(* IEC 61131-3 sources: LASAL/Class/ST151Base (part 2) *)

//**********************************************************************************************************************************************************
    _InitError:
      eModuleInitState := ERROR;
      if (eInitState <> _InvalidConfguration) then
        eInitState      := _ClientNotready;
      end_if;

//**********************************************************************************************************************************************************

  end_case;

END_FUNCTION

FUNCTION VIRTUAL GLOBAL ST151Base::GetDeviceID
	VAR_OUTPUT
		output 	: UDINT;
	END_VAR

  output := DEVICE_ID_ST151;

END_FUNCTION

FUNCTION VIRTUAL GLOBAL ST151Base::Enable::Write
	VAR_INPUT
		input (EAX) 	: DINT;
	END_VAR
	VAR_OUTPUT
		result (EAX) 	: DINT;
	END_VAR

  if input & AxError then
    input := 0;
  end_if;

  Enable := input;

  sAccesses.sWriteData.ControlWord.SwitchOn := ControlWord.SwitchOn := ControlWord.EnableOperation := to_bool(input);

  if input = 0 then
    SetFreqOut.Write(input:=0);
  end_if;

  result := Enable;

END_FUNCTION

FUNCTION VIRTUAL ST151Base::ReceiveSDOResponse
	VAR_INPUT
		eCommand 	: t_SDIAS_SDO_Cmd;
		hOffset 	: HINT;
		usLength 	: USINT;
		eResult 	: iprStates;
		pResponseBuffer 	: ^USINT;
		ResponseLength 	: USINT;
	END_VAR
	VAR_OUTPUT
		ret_code 	: iprStates;
	END_VAR

  ret_code := SdiasBase::ReceiveSDOResponse(eCommand, hOffset, usLength, eResult, pResponseBuffer, ResponseLength);

  // spi access from baseclass
  if bSDOResponseHandle = TRUE then
    return;
  end_if;

  if eResult = READY then

    case eCommand of
    //**********************************************************************
      SDIAS_SDO_CMD_MEM_WRITE:
        case hOffset of
        //-------------------------------------------------------------
          ST151_ADDR_SDO_1,
          ST151_ADDR_SDO_2,
          ST151_ADDR_SDO_5,
          ST151_ADDR_SDO_6:
            if eResponseState = _wait then
              eResponseState := _valid;
            end_if;
        end_case;

      //**************************************************************************************************************************
      SDIAS_SDO_CMD_MEM_READ:
        case hOffset of
          //***************************************************************************************************
          ST151_ADDR_SDO_1:
            if eResponseState = _wait then
              eResponseState := _valid;
              sReadSDO.SDOData1 := pResponseBuffer^$t_s_ConfigModule1;
            end_if;

          //***************************************************************************************************
          ST151_ADDR_SDO_2:
            if eResponseState = _wait then
              eResponseState := _valid;
              sReadSDO.SDOData2      := pResponseBuffer^$t_s_ConfigModule2;
            end_if;

          //***************************************************************************************************
          ST151_ADDR_SDO_3:
            if eResponseState = _wait then
              eResponseState := _valid;
              sReadSDO.SDOData3      := pResponseBuffer^$t_s_ConfigModule3;
            end_if;

          //***************************************************************************************************
          ST151_ADDR_SDO_4:
            if eResponseState = _wait then
              eResponseState := _valid;
              sReadSDO.SDOData4      := pResponseBuffer^$t_s_ConfigModule4;
            end_if;

          //***************************************************************************************************
          ST151_ADDR_SDO_5:
            if eResponseState = _wait then
              eResponseState := _valid;
              sReadSDO.SDOData5      := pResponseBuffer^$t_s_ConfigModule5;
            end_if;

          //***************************************************************************************************
          ST151_ADDR_SDO_6:
            if eResponseState = _wait then
              eResponseState := _valid;
              sReadSDO.SDOData6      := pResponseBuffer^$t_s_ConfigModule6;
            end_if;
        end_case;

      //**************************************************************************************************************************
      //Control Read
      SDIAS_SDO_CMD_CTRL_READ:
        if hOffset >= ST151_PLL_OFFSET
         & hOffset < (ST151_PLL_OFFSET+sizeof(sPllRegister)) then
          eResponseState := _valid;
          if eResponseState = _wait then
            _memcpy(ptr1:= (#sPllRegister + sSPIReadData.udReadOffset), ptr2:=pResponseBuffer, cntr:=sSPIReadData.udReadLength);
          end_if;
        end_if;

      //**************************************************************************************************************************
      //Control write
      SDIAS_SDO_CMD_CTRL_WRITE:
        if hOffset >= ST151_PLL_OFFSET
         & hOffset < (ST151_PLL_OFFSET+sizeof(sPllRegister)) then
          if eResponseState = _wait then
            eResponseState := _valid;
          end_if;
        end_if;

    end_case;

    if eResponseState <> _valid then
      LogError("@ZZZZ (ST151Base::ReceiveSDOResponse) ERROR in response data of SDO");
      // ERROR was at initialisation
      eInitSSW := _InitError;
    end_if;

  else
    case eCommand of
      SDIAS_SDO_CMD_MEM_WRITE:
        LogError("@ZZZZ (ST151Base::ReceiveSDOResponse) ERROR while writing the sdo data");
      SDIAS_SDO_CMD_MEM_READ:
        LogError("@ZZZZ (ST151Base::ReceiveSDOResponse) ERROR while reading the sdo data");
      SDIAS_SDO_CMD_CTRL_READ:
        LogError("@ZZZZ (ST151Base::ReceiveSDOResponse) Error while reading the pll configuration");
      SDIAS_SDO_CMD_CTRL_WRITE:
        LogError("@ZZZZ (ST151Base::ReceiveSDOResponse) Error while writing the pll configuration");
    end_case;
    // ERROR was at initialisation
    eInitSSW := _InitError;
  end_if;

END_FUNCTION

FUNCTION VIRTUAL GLOBAL ST151Base::Input1LatchedRising::Read
	VAR_OUTPUT
		output (EAX) 	: DINT;
	END_VAR

  //Return Latch
	output := Input1LatchedRising;

  //Reset Latch in next rt-run
  sLatchValues.bsLatchReaded.DigIn1Rise := TRUE;

END_FUNCTION

FUNCTION VIRTUAL GLOBAL ST151Base::Input1LatchedFalling::Read
	VAR_OUTPUT
		output (EAX) 	: DINT;
	END_VAR

  //Return Latch
	output := Input1LatchedFalling;

  //Reset Latch in next rt-run
  sLatchValues.bsLatchReaded.DigIn1Fall := TRUE;

END_FUNCTION

FUNCTION VIRTUAL GLOBAL ST151Base::Input2LatchedRising::Read
	VAR_OUTPUT
		output (EAX) 	: DINT;
	END_VAR

  //Return Latch
	output := Input2LatchedRising;

  //Reset Latch in next rt-run
  sLatchValues.bsLatchReaded.DigIn2Rise := TRUE;

END_FUNCTION

FUNCTION VIRTUAL GLOBAL ST151Base::Input2LatchedFalling::Read
	VAR_OUTPUT
		output (EAX) 	: DINT;
	END_VAR

  //Return Latch
	output := Input2LatchedFalling;

  //Reset Latch in next rt-run
  sLatchValues.bsLatchReaded.DigIn2Fall := TRUE;

END_FUNCTION

FUNCTION VIRTUAL GLOBAL ST151Base::ZPulsLatched::Read
	VAR_OUTPUT
		output (EAX) 	: DINT;
	END_VAR

  //Return Latch
	output := ZPulsLatched;

  //Reset Latch in next rt-run
  sLatchValues.bsLatchReaded.IncZero := TRUE;

END_FUNCTION

FUNCTION VIRTUAL GLOBAL ST151Base::DisconnectEvent
  //Reset DO-Data
  if sAccesses.pWriteData then
    _memset(dest := sAccesses.pWriteData, usByte := 0, cntr := sizeof(sAccesses.pWriteData^));
  end_if;

  //reset online state
  Online  := 0;

  //Call Disconnect of Base-Class
  SdiasBase::DisconnectEvent();

END_FUNCTION

FUNCTION ST151Base::ST151Base
	VAR_OUTPUT
		ret_code 	: ConfStates;
	END_VAR

	ret_code := C_OK;

END_FUNCTION

FUNCTION VIRTUAL ST151Base::GetTaskCfg
	VAR_OUTPUT
		TaskCfg 	: BDINT;
	END_VAR

  TaskCfg := SDIAS_TASK_MASK_RT_PRE OR SDIAS_TASK_MASK_RT_POST OR SDIAS_TASK_MASK_CY;

END_FUNCTION

FUNCTION VIRTUAL GLOBAL ST151Base::ErrorQuit::Write
	VAR_INPUT
		input (EAX) 	: DINT;
	END_VAR
	VAR_OUTPUT
		result (EAX) 	: DINT;
	END_VAR

  result := ErrorQuit := sAccesses.sWriteData.ControlWord.RegenResistorFaultReset := sAccesses.sWriteData.ControlWord.QuitSTOOff := sAccesses.sWriteData.ControlWord.FaultReset := ControlWord.ResetFault := to_bool(input);

END_FUNCTION

FUNCTION VIRTUAL GLOBAL ST151Base::CurrentIncrease::Write
	VAR_INPUT
		input (EAX) 	: DINT;
	END_VAR
	VAR_OUTPUT
		result (EAX) 	: DINT;
	END_VAR

  result := CurrentIncrease := sAccesses.sWriteData.ControlWord.CurrentIncrease := ControlWord.ManufactureSpec1 := to_bool(input);

END_FUNCTION

FUNCTION VIRTUAL GLOBAL ST151Base::ControlWord::Write
	VAR_INPUT
		input (EAX) 	: DS402_Control;
	END_VAR
	VAR_OUTPUT
		result (EAX) 	: DS402_Control;
	END_VAR

  result := ControlWord := input;

  Enable := ControlWord.SwitchOn AND ControlWord.EnableOperation;
  sAccesses.sWriteData.ControlWord.SwitchOn   := to_BOOL(Enable);
  sAccesses.sWriteData.ControlWord.FaultReset := sAccesses.sWriteData.ControlWord.RegenResistorFaultReset := sAccesses.sWriteData.ControlWord.QuitSTOOff := ControlWord.ResetFault;
  CurrentIncrease := sAccesses.sWriteData.ControlWord.CurrentIncrease := ControlWord.ManufactureSpec1;

END_FUNCTION

FUNCTION VIRTUAL GLOBAL ST151Base::SetFreqOut::Write
	VAR_INPUT
		input (EAX) 	: DINT;
	END_VAR
	VAR_OUTPUT
		result (EAX) 	: DINT;
	END_VAR
  VAR
  	dTempInput : DINT;
  END_VAR

  if input <> SetFreqOut then //just do something when the value changed
    dTempInput := input * usCompModeVST;
    if dTempInput > ST151_MAXFREQUENCY_OUT then
      dTempInput := ST151_MAXFREQUENCY_OUT;
    elsif dTempInput < -ST151_MAXFREQUENCY_OUT then
      dTempInput := -ST151_MAXFREQUENCY_OUT;
    end_if;

    //*****************************************************************************
    SetFreqOut := input;

    //Calculate Current
    sAccesses.sWriteData.ControlWord.SwitchMaxCurrent := (abs(input)$UDINT <= udStallCurrentWindow);
    //write act frequency to module
    sAccesses.sWriteData.StepFrequencyReg := dTempInput;

  end_if;

  result := SetFreqOut;

END_FUNCTION

FUNCTION VIRTUAL GLOBAL ST151Base::TargetFreqOut::Write
	VAR_INPUT
		input (EAX) 	: DINT;
	END_VAR
	VAR_OUTPUT
		result (EAX) 	: DINT;
	END_VAR
  VAR
  	dRetCode : DINT;
  END_VAR

  // calculate adaptive microstepping
	TargetFreqOut := input;
  if TargetFreqOut <> -1 then
    //calculate always from zero to target frequency
    dRetCode       := CalcAdaptiveMicroStepping(dTargetFrequency:=TargetFreqOut, dActSetFrequency:=0);
  else
    EnableSteps.Write(input:=EnableSteps+0x800); // +0x800 is just to have a change of the value. It is rejected inside the write()
  end_if;

  if dRetCode = 0 then
    //all ok write setting
  end_if;
	result         := TargetFreqOut;

END_FUNCTION

FUNCTION VIRTUAL GLOBAL ST151Base::HWRampdownDeltaFrequency::Write
	VAR_INPUT
		input (EAX) 	: DINT;
	END_VAR
	VAR_OUTPUT
		result (EAX) 	: DINT;
	END_VAR

  sWriteSDO.SDOData2.HWRampdownDeltaFrequency := input$UINT;
  biReqSDOConfigRdWr.WriteConfigSDO2          := TRUE;
  HWRampdownDeltaFrequency := input;
  result                   := HWRampdownDeltaFrequency;

END_FUNCTION

FUNCTION VIRTUAL GLOBAL ST151Base::HWRampdownDeltaTime::Write
	VAR_INPUT
		input (EAX) 	: DINT;
	END_VAR
	VAR_OUTPUT
		result (EAX) 	: DINT;
	END_VAR

  sWriteSDO.SDOData2.HWRampdownDeltaTime := input$uint;
  biReqSDOConfigRdWr.WriteConfigSDO2     := TRUE;
  HWRampdownDeltaTime := input;
  result              := HWRampdownDeltaTime;

END_FUNCTION

FUNCTION VIRTUAL GLOBAL ST151Base::HWEnableSoftwareRampdown::Write
	VAR_INPUT
		input (EAX) 	: DINT;
	END_VAR
	VAR_OUTPUT
		result (EAX) 	: DINT;
	END_VAR

  HWEnableSoftwareRampdown := input <> 0;
 	result := HWEnableSoftwareRampdown;

END_FUNCTION

FUNCTION ST151Base::SDORdWrData
	VAR_OUTPUT
		dRetCode 	: iprStates;
	END_VAR
  VAR
  	TmpRetcode : iprStates;
  END_VAR

  dRetCode := BUSY;

  case eActSDOConfigRdWr of
    //********************************************************************************************************************************
  	t_e_SDOConfig::_SDOConfig_Idle:
      eActSDOConfigRdWr := SetSDORdWrStep(eActStep:=eActSDOConfigRdWr);

    //********************************************************************************************************************************
  	t_e_SDOConfig::_SDOConfig_Write1:
      case eResponseState of
        _idle:
          biReqSDOConfigRdWr.WriteConfigSDO1  := FALSE;
          bsRespSDOConfigRdWr.WriteConfigSDO1 := FALSE;
          TmpRetcode  := StartWriteSDO(hOffset:=ST151_ADDR_SDO_1, usLength:=sizeof(sWriteSDO.SDOData1), pWriteBuffer:=(#sWriteSDO.SDOData1)$^USINT, eCommand:=SDIAS_SDO_CMD_MEM_WRITE);
          if TmpRetcode = READY then
            udSDOTimeout  := ops.tAbsolute;
            eResponseState:= _wait;
          elsif TmpRetcode = ERROR then
            LogError("@ZZZZ (ST151Base::SDORdWrData) Failed to add write SDO for configuration");
            eActSDOConfigRdWr := _SDOConfig_Error;
          end_if;
          //*****************************************************
        _wait:
          // wait for response
          if ((ops.tAbsolute - udSDOTimeout) > ST151_SDO_RESPONSE_TIMEOUT) then
            LogError("@ZZZZ (ST151Base::SDORdWrData) SDO Response timeout config module");
            eActSDOConfigRdWr := _SDOConfig_Error;
          end_if;
        //*****************************************************
        _valid:
          eActSDOConfigRdWr := SetSDORdWrStep(eActStep:=eActSDOConfigRdWr);
          bsRespSDOConfigRdWr.WriteConfigSDO1 := TRUE;
          eResponseState                      := _idle;
        //*****************************************************
      end_case;

    //********************************************************************************************************************************
  	t_e_SDOConfig::_SDOConfig_Write2:
      case eResponseState of
        _idle:
          biReqSDOConfigRdWr.WriteConfigSDO2  := FALSE;
          bsRespSDOConfigRdWr.WriteConfigSDO2 := FALSE;
          TmpRetcode  := StartWriteSDO(hOffset:=ST151_ADDR_SDO_2, usLength:=sizeof(sWriteSDO.SDOData2), pWriteBuffer:=(#sWriteSDO.SDOData2)$^USINT, eCommand:=SDIAS_SDO_CMD_MEM_WRITE);
          if TmpRetcode = READY then
            udSDOTimeout  := ops.tAbsolute;
            eResponseState:= _wait;
          elsif TmpRetcode = ERROR then
            LogError("@ZZZZ (ST151Base::SDORdWrData) Failed to add write SDO for configuration");
            eActSDOConfigRdWr := _SDOConfig_Error;
          end_if;
          //*****************************************************
        _wait:
          // wait for response
          if ((ops.tAbsolute - udSDOTimeout) > ST151_SDO_RESPONSE_TIMEOUT) then
            LogError("@ZZZZ (ST151Base::SDORdWrData) SDO Response timeout config module");
            eActSDOConfigRdWr := _SDOConfig_Error;
          end_if;
        //*****************************************************
        _valid:
          eActSDOConfigRdWr := SetSDORdWrStep(eActStep:=eActSDOConfigRdWr);
          bsRespSDOConfigRdWr.WriteConfigSDO2 := TRUE;
          eResponseState                      := _idle;
        //*****************************************************
      end_case;

    //********************************************************************************************************************************
  	t_e_SDOConfig::_SDOConfig_Write3:
      //sdo 3 is only read
//      case eResponseState of
//        _idle:
          biReqSDOConfigRdWr.WriteConfigSDO3  := FALSE;
          bsRespSDOConfigRdWr.WriteConfigSDO3 := FALSE;
//          TmpRetcode  := StartWriteSDO(hOffset:=ST151_ADDR_SDO_3, usLength:=sizeof(sWriteSDO.SDOData3), pWriteBuffer:=(#sWriteSDO.SDOData3)$^USINT, eCommand:=SDIAS_SDO_CMD_MEM_WRITE);
//          if TmpRetcode = READY then
//            udSDOTimeout  := ops.tAbsolute;
//            eResponseState:= _wait;
//          elsif TmpRetcode = ERROR then
//            LogError("@ZZZZ (ST151Base::SDORdWrData) Failed to add write SDO for configuration");
//            eActSDOConfigRdWr := _SDOConfig_Error;
//          end_if;
//          //*****************************************************
//        _wait:
//          // wait for response
//          if ((ops.tAbsolute - udSDOTimeout) > ST151_SDO_RESPONSE_TIMEOUT) then
//            LogError("@ZZZZ (ST151Base::SDORdWrData) SDO Response timeout config module");
//            eActSDOConfigRdWr := _SDOConfig_Error;
//          end_if;
//        //*****************************************************
//        _valid:
          eActSDOConfigRdWr := SetSDORdWrStep(eActStep:=eActSDOConfigRdWr);
//          bsRespSDOConfigRdWr.WriteConfigSDO3 := TRUE;
//          eResponseState                      := _idle;
//        //*****************************************************
//      end_case;

    //********************************************************************************************************************************
  	t_e_SDOConfig::_SDOConfig_Write4:
      //sdo 4 is only read
//      case eResponseState of
//        _idle:
          biReqSDOConfigRdWr.WriteConfigSDO4  := FALSE;
          bsRespSDOConfigRdWr.WriteConfigSDO4 := FALSE;
//          TmpRetcode  := StartWriteSDO(hOffset:=ST151_ADDR_SDO_4, usLength:=sizeof(sWriteSDO.SDOData4), pWriteBuffer:=(#sWriteSDO.SDOData4)$^USINT, eCommand:=SDIAS_SDO_CMD_MEM_WRITE);
//          if TmpRetcode = READY then
//            udSDOTimeout  := ops.tAbsolute;
//            eResponseState:= _wait;
//          elsif TmpRetcode = ERROR then
//            LogError("@ZZZZ (ST151Base::SDORdWrData) Failed to add write SDO for configuration");
//            eActSDOConfigRdWr := _SDOConfig_Error;
//          end_if;
//          //*****************************************************
//        _wait:
//          // wait for response
//          if ((ops.tAbsolute - udSDOTimeout) > ST151_SDO_RESPONSE_TIMEOUT) then
//            LogError("@ZZZZ (ST151Base::SDORdWrData) SDO Response timeout config module");
//            eActSDOConfigRdWr := _SDOConfig_Error;
//          end_if;
//        //*****************************************************
//        _valid:
          eActSDOConfigRdWr := SetSDORdWrStep(eActStep:=eActSDOConfigRdWr);
//          bsRespSDOConfigRdWr.WriteConfigSDO4 := TRUE;
//          eResponseState                      := _idle;
//        //*****************************************************
//      end_case;

    //********************************************************************************************************************************
  	t_e_SDOConfig::_SDOConfig_Write5:
      case eResponseState of
        _idle:
          biReqSDOConfigRdWr.WriteConfigSDO5  := FALSE;
          bsRespSDOConfigRdWr.WriteConfigSDO5 := FALSE;
          TmpRetcode  := StartWriteSDO(hOffset:=ST151_ADDR_SDO_5, usLength:=sizeof(sWriteSDO.SDOData5), pWriteBuffer:=(#sWriteSDO.SDOData5)$^USINT, eCommand:=SDIAS_SDO_CMD_MEM_WRITE);
          if TmpRetcode = READY then
            udSDOTimeout  := ops.tAbsolute;
            eResponseState:= _wait;
          elsif TmpRetcode = ERROR then
            LogError("@ZZZZ (ST151Base::SDORdWrData) Failed to add write SDO for configuration");
            eActSDOConfigRdWr := _SDOConfig_Error;
          end_if;
          //*****************************************************
        _wait:
          // wait for response
          if ((ops.tAbsolute - udSDOTimeout) > ST151_SDO_RESPONSE_TIMEOUT) then
            LogError("@ZZZZ (ST151Base::SDORdWrData) SDO Response timeout config module");
            eActSDOConfigRdWr := _SDOConfig_Error;
          end_if;
        //*****************************************************
        _valid:
          eActSDOConfigRdWr := SetSDORdWrStep(eActStep:=eActSDOConfigRdWr);
          bsRespSDOConfigRdWr.WriteConfigSDO5 := TRUE;
          eResponseState                      := _idle;
        //*****************************************************
      end_case;

    //********************************************************************************************************************************
  	t_e_SDOConfig::_SDOConfig_Write6:
      case eResponseState of
        _idle:
          biReqSDOConfigRdWr.WriteConfigSDO6  := FALSE;
          bsRespSDOConfigRdWr.WriteConfigSDO6 := FALSE;
          TmpRetcode  := StartWriteSDO(hOffset:=ST151_ADDR_SDO_6, usLength:=sizeof(sWriteSDO.SDOData6), pWriteBuffer:=(#sWriteSDO.SDOData6)$^USINT, eCommand:=SDIAS_SDO_CMD_MEM_WRITE);
          if TmpRetcode = READY then
            udSDOTimeout  := ops.tAbsolute;
            eResponseState:= _wait;
          elsif TmpRetcode = ERROR then
            LogError("@ZZZZ (ST151Base::SDORdWrData) Failed to add write SDO for configuration");
            eActSDOConfigRdWr := _SDOConfig_Error;
          end_if;
          //*****************************************************
        _wait:
          // wait for response
          if ((ops.tAbsolute - udSDOTimeout) > ST151_SDO_RESPONSE_TIMEOUT) then
            LogError("@ZZZZ (ST151Base::SDORdWrData) SDO Response timeout config module");
            eActSDOConfigRdWr := _SDOConfig_Error;
          end_if;
        //*****************************************************
        _valid:
          eActSDOConfigRdWr := SetSDORdWrStep(eActStep:=eActSDOConfigRdWr);
          bsRespSDOConfigRdWr.WriteConfigSDO6 := TRUE;
          eResponseState                      := _idle;
        //*****************************************************
      end_case;

    //********************************************************************************************************************************
  	t_e_SDOConfig::_SDOConfig_Read1:
      case eResponseState of
        _idle:
          biReqSDOConfigRdWr.ReadConfigSDO1  := FALSE;
          bsRespSDOConfigRdWr.ReadConfigSDO1 := FALSE;
          TmpRetcode  := StartReadSDO(hOffset:=ST151_ADDR_SDO_1, usLength:=sizeof(sReadSDO.SDOData1), eCommand:=SDIAS_SDO_CMD_MEM_READ);
          if TmpRetcode = READY then
            udSDOTimeout  := ops.tAbsolute;
            eResponseState:= _wait;
          elsif TmpRetcode = ERROR then
            LogError("@ZZZZ (ST151Base::SDORdWrData) Failed to add SDO for read of configuration");
            eActSDOConfigRdWr := _SDOConfig_Error;
          end_if;
          //*****************************************************
        _wait:
          // wait for response
          if ((ops.tAbsolute - udSDOTimeout) > ST151_SDO_RESPONSE_TIMEOUT) then
            LogError("@ZZZZ (ST151Base::SDORdWrData) SDO Response timeout config module");
            eActSDOConfigRdWr := _SDOConfig_Error;
          end_if;
        //*****************************************************
        _valid:
          eActSDOConfigRdWr := SetSDORdWrStep(eActStep:=eActSDOConfigRdWr);
          bsRespSDOConfigRdWr.ReadConfigSDO1  := TRUE;
          eResponseState                      := _idle;
        //*****************************************************
      end_case;

    //********************************************************************************************************************************
  	t_e_SDOConfig::_SDOConfig_Read2:
      case eResponseState of
        _idle:
          biReqSDOConfigRdWr.ReadConfigSDO2  := FALSE;
          bsRespSDOConfigRdWr.ReadConfigSDO2 := FALSE;
          TmpRetcode  := StartReadSDO(hOffset:=ST151_ADDR_SDO_2, usLength:=sizeof(sReadSDO.SDOData2), eCommand:=SDIAS_SDO_CMD_MEM_READ);
          if TmpRetcode = READY then
            udSDOTimeout  := ops.tAbsolute;
            eResponseState:= _wait;
          elsif TmpRetcode = ERROR then
            LogError("@ZZZZ (ST151Base::SDORdWrData) Failed to add SDO for read of configuration");
            eActSDOConfigRdWr := _SDOConfig_Error;
          end_if;
          //*****************************************************
        _wait:
          // wait for response
          if ((ops.tAbsolute - udSDOTimeout) > ST151_SDO_RESPONSE_TIMEOUT) then
            LogError("@ZZZZ (ST151Base::SDORdWrData) SDO Response timeout config module");
            eActSDOConfigRdWr := _SDOConfig_Error;
          end_if;
        //*****************************************************
        _valid:
          eActSDOConfigRdWr := SetSDORdWrStep(eActStep:=eActSDOConfigRdWr);
          bsRespSDOConfigRdWr.ReadConfigSDO2  := TRUE;
          eResponseState                      := _idle;
        //*****************************************************
      end_case;

    //********************************************************************************************************************************
  	t_e_SDOConfig::_SDOConfig_Read3:
      case eResponseState of
        _idle:
          biReqSDOConfigRdWr.ReadConfigSDO3  := FALSE;
          bsRespSDOConfigRdWr.ReadConfigSDO3 := FALSE;
          TmpRetcode  := StartReadSDO(hOffset:=ST151_ADDR_SDO_3, usLength:=sizeof(sReadSDO.SDOData3), eCommand:=SDIAS_SDO_CMD_MEM_READ);
          if TmpRetcode = READY then
            //save the actual latched values
            sLatchValues.bsValidISyncValue     := sLatchValues.bsActiveISyncValue;
            sLatchValues.bResetActiveSyncValue := TRUE;
            udSDOTimeout  := ops.tAbsolute;
            eResponseState:= _wait;
          elsif TmpRetcode = ERROR then
            LogError("@ZZZZ (ST151Base::SDORdWrData) Failed to add SDO for read of configuration");
            eActSDOConfigRdWr := _SDOConfig_Error;
          end_if;
          //*****************************************************
        _wait:
          // wait for response
          if ((ops.tAbsolute - udSDOTimeout) > ST151_SDO_RESPONSE_TIMEOUT) then
            LogError("@ZZZZ (ST151Base::SDORdWrData) SDO Response timeout config module");
            eActSDOConfigRdWr := _SDOConfig_Error;
          end_if;
        //*****************************************************
        _valid:
          eActSDOConfigRdWr := SetSDORdWrStep(eActStep:=eActSDOConfigRdWr);
          bsRespSDOConfigRdWr.ReadConfigSDO3  := TRUE;
          eResponseState                      := _idle;
        //*****************************************************
      end_case;

    //********************************************************************************************************************************
  	t_e_SDOConfig::_SDOConfig_Read4:
      case eResponseState of
        _idle:
          biReqSDOConfigRdWr.ReadConfigSDO4  := FALSE;
          bsRespSDOConfigRdWr.ReadConfigSDO4 := FALSE;
          TmpRetcode  := StartReadSDO(hOffset:=ST151_ADDR_SDO_4, usLength:=sizeof(sReadSDO.SDOData4), eCommand:=SDIAS_SDO_CMD_MEM_READ);
          if TmpRetcode = READY then
            //save the actual latched values
            sLatchValues.bsValidISyncValue     := sLatchValues.bsActiveISyncValue;
            sLatchValues.bResetActiveSyncValue := TRUE;
            udSDOTimeout  := ops.tAbsolute;
            eResponseState:= _wait;
          elsif TmpRetcode = ERROR then
            LogError("@ZZZZ (ST151Base::SDORdWrData) Failed to add SDO for read of configuration");
            eActSDOConfigRdWr := _SDOConfig_Error;
          end_if;
          //*****************************************************
        _wait:
          // wait for response
          if ((ops.tAbsolute - udSDOTimeout) > ST151_SDO_RESPONSE_TIMEOUT) then
            LogError("@ZZZZ (ST151Base::SDORdWrData) SDO Response timeout config module");
            eActSDOConfigRdWr := _SDOConfig_Error;
          end_if;
        //*****************************************************
        _valid:
          eActSDOConfigRdWr := SetSDORdWrStep(eActStep:=eActSDOConfigRdWr);
          bsRespSDOConfigRdWr.ReadConfigSDO4  := TRUE;
          eResponseState                      := _idle;
        //*****************************************************
      end_case;

    //********************************************************************************************************************************
  	t_e_SDOConfig::_SDOConfig_Read5:
      case eResponseState of
        _idle:
          biReqSDOConfigRdWr.ReadConfigSDO5  := FALSE;
          bsRespSDOConfigRdWr.ReadConfigSDO5 := FALSE;
          TmpRetcode  := StartReadSDO(hOffset:=ST151_ADDR_SDO_5, usLength:=sizeof(sReadSDO.SDOData5), eCommand:=SDIAS_SDO_CMD_MEM_READ);
          if TmpRetcode = READY then
            udSDOTimeout  := ops.tAbsolute;
            eResponseState:= _wait;
          elsif TmpRetcode = ERROR then
            LogError("@ZZZZ (ST151Base::SDORdWrData) Failed to add SDO for read of configuration");
            eActSDOConfigRdWr := _SDOConfig_Error;
          end_if;
          //*****************************************************
        _wait:
          // wait for response
          if ((ops.tAbsolute - udSDOTimeout) > ST151_SDO_RESPONSE_TIMEOUT) then
            LogError("@ZZZZ (ST151Base::SDORdWrData) SDO Response timeout config module");
            eActSDOConfigRdWr := _SDOConfig_Error;
          end_if;
        //*****************************************************
        _valid:
          eActSDOConfigRdWr := SetSDORdWrStep(eActStep:=eActSDOConfigRdWr);
          bsRespSDOConfigRdWr.ReadConfigSDO5  := TRUE;
          eResponseState                      := _idle;
        //*****************************************************
      end_case;

    //********************************************************************************************************************************
  	t_e_SDOConfig::_SDOConfig_Read6:
      case eResponseState of
        _idle:
          biReqSDOConfigRdWr.ReadConfigSDO6  := FALSE;
          bsRespSDOConfigRdWr.ReadConfigSDO6 := FALSE;
          TmpRetcode  := StartReadSDO(hOffset:=ST151_ADDR_SDO_6, usLength:=sizeof(sReadSDO.SDOData6), eCommand:=SDIAS_SDO_CMD_MEM_READ);
          if TmpRetcode = READY then
            udSDOTimeout  := ops.tAbsolute;
            eResponseState:= _wait;
          elsif TmpRetcode = ERROR then
            LogError("@ZZZZ (ST151Base::SDORdWrData) Failed to add SDO for read of configuration");
            eActSDOConfigRdWr := _SDOConfig_Error;
          end_if;
          //*****************************************************
        _wait:
          // wait for response
          if ((ops.tAbsolute - udSDOTimeout) > ST151_SDO_RESPONSE_TIMEOUT) then
            LogError("@ZZZZ (ST151Base::SDORdWrData) SDO Response timeout config module");
            eActSDOConfigRdWr := _SDOConfig_Error;
          end_if;
        //*****************************************************
        _valid:
          eActSDOConfigRdWr := SetSDORdWrStep(eActStep:=eActSDOConfigRdWr);
          bsRespSDOConfigRdWr.ReadConfigSDO6  := TRUE;
          eResponseState                      := _idle;
        //*****************************************************
      end_case;

    //********************************************************************************************************************************
  	t_e_SDOConfig::_SDOConfig_Finished:
      //all ok sdo config is finished
      dRetCode          := READY;
      usSDORetrys       := 0;
      eActSDOConfigRdWr := _SDOConfig_Idle;

    //********************************************************************************************************************************
  	t_e_SDOConfig::_SDOConfig_Error:
      dRetCode          := ERROR;
      usSDORetrys       += 1;
      if usSDORetrys < ST151_SDO_MAX_RETRYS then
        eActSDOConfigRdWr := _SDOConfig_Idle;
      end_if;
      eResponseState    := _idle;

  end_case;

END_FUNCTION

FUNCTION VIRTUAL GLOBAL ST151Base::FrequLimitIncrease2to1::Write
	VAR_INPUT
		input (EAX) 	: UDINT;
	END_VAR
	VAR_OUTPUT
		result (EAX) 	: UDINT;
	END_VAR
  VAR
    siActArrayEntry : SINT;
  END_VAR

  siActArrayEntry := 0;
  //calculate compatibility mode if client is set
  input *= usCompModeVST;

   // Check for max frequency limit
  if input > ST151_MAXFREQUENCY_OUT then
    input := ST151_MAXFREQUENCY_OUT;
  end_if;

  if aFrequencyLimit[siActArrayEntry].LimitIncrease <> input then //do we have a new value?
    //Save Input
    FrequLimitIncrease2to1 := input / usCompModeVST;

    aFrequencyLimit[siActArrayEntry].LimitIncrease := input;
    FrequLimitDecrease1to2.Write(input:=FrequLimitDecrease1to2);

    if aFrequencyLimit[siActArrayEntry].LimitIncrease <> sWriteSDO.SDOData1.FrequLimitRising2 then //do we have a new value?
      //Set new Limit
      sWriteSDO.SDOData1.FrequLimitRising2 := aFrequencyLimit[siActArrayEntry].LimitIncrease;
      biReqSDOConfigRdWr.WriteConfigSDO1   := TRUE;
    end_if;
  end_if;

  result := FrequLimitIncrease2to1;

END_FUNCTION

FUNCTION VIRTUAL GLOBAL ST151Base::FrequLimitIncrease4to2::Write
	VAR_INPUT
		input (EAX) 	: UDINT;
	END_VAR
	VAR_OUTPUT
		result (EAX) 	: UDINT;
	END_VAR
  VAR
    siActArrayEntry : SINT;
  END_VAR

  siActArrayEntry := 1;
  //calculate compatibility mode if client is set
  input *= usCompModeVST;

   // Check for max frequency limit
  if input > ST151_MAXFREQUENCY_OUT then
    input := ST151_MAXFREQUENCY_OUT;
  end_if;

  if aFrequencyLimit[siActArrayEntry].LimitIncrease <> input then //do we have a new value?
    //Save Input
    FrequLimitIncrease4to2 := input / usCompModeVST;

    aFrequencyLimit[siActArrayEntry].LimitIncrease := input;
    FrequLimitDecrease2to4.Write(input:=FrequLimitDecrease2to4);

    if aFrequencyLimit[siActArrayEntry].LimitIncrease <> sWriteSDO.SDOData1.FrequLimitRising4 then //do we have a new value?
      //Set new Limit
      sWriteSDO.SDOData1.FrequLimitRising4 := aFrequencyLimit[siActArrayEntry].LimitIncrease;
      biReqSDOConfigRdWr.WriteConfigSDO1   := TRUE;
    end_if;
  end_if;

  result := FrequLimitIncrease4to2;

END_FUNCTION

FUNCTION VIRTUAL GLOBAL ST151Base::FrequLimitIncrease8to4::Write
	VAR_INPUT
		input (EAX) 	: UDINT;
	END_VAR
	VAR_OUTPUT
		result (EAX) 	: UDINT;
	END_VAR
  VAR
    siActArrayEntry : SINT;
  END_VAR

  siActArrayEntry := 2;
  //calculate compatibility mode if client is set
  input *= usCompModeVST;

   // Check for max frequency limit
  if input > ST151_MAXFREQUENCY_OUT then
    input := ST151_MAXFREQUENCY_OUT;
  end_if;

  if aFrequencyLimit[siActArrayEntry].LimitIncrease <> input then //do we have a new value?
    //Save Input
    FrequLimitIncrease8to4 := input / usCompModeVST;

    aFrequencyLimit[siActArrayEntry].LimitIncrease := input;
    FrequLimitDecrease4to8.Write(input:=FrequLimitDecrease4to8);

    if aFrequencyLimit[siActArrayEntry].LimitIncrease <> sWriteSDO.SDOData1.FrequLimitRising8 then //do we have a new value?
      //Set new Limit
      sWriteSDO.SDOData1.FrequLimitRising8 := aFrequencyLimit[siActArrayEntry].LimitIncrease;
      biReqSDOConfigRdWr.WriteConfigSDO1   := TRUE;
    end_if;
  end_if;

  result := FrequLimitIncrease8to4;

END_FUNCTION

FUNCTION VIRTUAL GLOBAL ST151Base::FrequLimitIncrease16to8::Write
	VAR_INPUT
		input (EAX) 	: UDINT;
	END_VAR
	VAR_OUTPUT
		result (EAX) 	: UDINT;
	END_VAR
  VAR
    siActArrayEntry : SINT;
  END_VAR

  siActArrayEntry := 3;
  //calculate compatibility mode if client is set
  input *= usCompModeVST;

   // Check for max frequency limit
  if input > ST151_MAXFREQUENCY_OUT then
    input := ST151_MAXFREQUENCY_OUT;
  end_if;

  if aFrequencyLimit[siActArrayEntry].LimitIncrease <> input then //do we have a new value?
    //Save Input
    FrequLimitIncrease16to8 := input / usCompModeVST;

    aFrequencyLimit[siActArrayEntry].LimitIncrease := input;
    FrequLimitDecrease8to16.Write(input:=FrequLimitDecrease8to16);

    if aFrequencyLimit[siActArrayEntry].LimitIncrease <> sWriteSDO.SDOData1.FrequLimitRising16 then //do we have a new value?
      //Set new Limit
      sWriteSDO.SDOData1.FrequLimitRising16 := aFrequencyLimit[siActArrayEntry].LimitIncrease;
      biReqSDOConfigRdWr.WriteConfigSDO1    := TRUE;
    end_if;
  end_if;

  result := FrequLimitIncrease16to8;

END_FUNCTION

FUNCTION VIRTUAL GLOBAL ST151Base::FrequLimitIncrease32to16::Write
	VAR_INPUT
		input (EAX) 	: UDINT;
	END_VAR
	VAR_OUTPUT
		result (EAX) 	: UDINT;
	END_VAR
  VAR
    siActArrayEntry : SINT;
  END_VAR

  siActArrayEntry := 4;
  //calculate compatibility mode if client is set
  input *= usCompModeVST;

   // Check for max frequency limit
  if input > ST151_MAXFREQUENCY_OUT then
    input := ST151_MAXFREQUENCY_OUT;
  end_if;

  if aFrequencyLimit[siActArrayEntry].LimitIncrease <> input then //do we have a new value?
    //Save Input
    FrequLimitIncrease32to16 := input / usCompModeVST;

    aFrequencyLimit[siActArrayEntry].LimitIncrease := input;
    FrequLimitDecrease16to32.Write(input:=FrequLimitDecrease16to32);

    if aFrequencyLimit[siActArrayEntry].LimitIncrease <> sWriteSDO.SDOData1.FrequLimitRising32 then //do we have a new value?
      //Set new Limit
      sWriteSDO.SDOData1.FrequLimitRising32 := aFrequencyLimit[siActArrayEntry].LimitIncrease;
      biReqSDOConfigRdWr.WriteConfigSDO1    := TRUE;
    end_if;
  end_if;

  result := FrequLimitIncrease32to16;

END_FUNCTION

FUNCTION VIRTUAL GLOBAL ST151Base::FrequLimitIncrease64to32::Write
	VAR_INPUT
		input (EAX) 	: UDINT;
	END_VAR
	VAR_OUTPUT
		result (EAX) 	: UDINT;
	END_VAR
  VAR
    siActArrayEntry : SINT;
  END_VAR

  siActArrayEntry := 5;
  //calculate compatibility mode if client is set
  input *= usCompModeVST;

   // Check for max frequency limit
  if input > ST151_MAXFREQUENCY_OUT then
    input := ST151_MAXFREQUENCY_OUT;
  end_if;

  if aFrequencyLimit[siActArrayEntry].LimitIncrease <> input then //do we have a new value?
    //Save Input
    FrequLimitIncrease64to32 := input / usCompModeVST;

    aFrequencyLimit[siActArrayEntry].LimitIncrease := input;
    FrequLimitDecrease32to64.Write(input:=FrequLimitDecrease32to64);

    if aFrequencyLimit[siActArrayEntry].LimitIncrease <> sWriteSDO.SDOData1.FrequLimitRising64 then //do we have a new value?
      //Set new Limit
      sWriteSDO.SDOData1.FrequLimitRising64 := aFrequencyLimit[siActArrayEntry].LimitIncrease;
      biReqSDOConfigRdWr.WriteConfigSDO1    := TRUE;
    end_if;
  end_if;

  result := FrequLimitIncrease64to32;

END_FUNCTION

FUNCTION VIRTUAL GLOBAL ST151Base::FrequLimitDecrease1to2::Write
	VAR_INPUT
		input (EAX) 	: UDINT;
	END_VAR
	VAR_OUTPUT
		result (EAX) 	: UDINT;
	END_VAR
  VAR
    siActArrayEntry : SINT;
  END_VAR

  siActArrayEntry := 0;
  //calculate compatibility mode if client is set
  input *= usCompModeVST;

   // Check for max frequency limit
  if input > ST151_MAXFREQUENCY_OUT then
    input := ST151_MAXFREQUENCY_OUT;
  end_if;
  //Save Input
  FrequLimitDecrease1to2 := input / usCompModeVST;

  if input <> ST151_AUTOSET_FREQUENCYLIMIT then
    aFrequencyLimit[siActArrayEntry].LimitDecrease := input;
  else
    CalcSimpleMode();
  end_if;

  if aFrequencyLimit[siActArrayEntry].LimitDecrease <> sWriteSDO.SDOData5.FrequLimitFalling1to2 then //do we have a new value?
    //Set new Limit
    sWriteSDO.SDOData5.FrequLimitFalling1to2 := aFrequencyLimit[siActArrayEntry].LimitDecrease;
    biReqSDOConfigRdWr.WriteConfigSDO5       := TRUE;
  end_if;

  result := FrequLimitDecrease1to2;

END_FUNCTION

FUNCTION VIRTUAL GLOBAL ST151Base::FrequLimitDecrease2to4::Write
	VAR_INPUT
		input (EAX) 	: UDINT;
	END_VAR
	VAR_OUTPUT
		result (EAX) 	: UDINT;
	END_VAR
  VAR
    siActArrayEntry : SINT;
  END_VAR

  siActArrayEntry := 1;
  //calculate compatibility mode if client is set
  input *= usCompModeVST;

   // Check for max frequency limit
  if input > ST151_MAXFREQUENCY_OUT then
    input := ST151_MAXFREQUENCY_OUT;
  end_if;
  //Save Input
  FrequLimitDecrease2to4 := input / usCompModeVST;

  if input <> ST151_AUTOSET_FREQUENCYLIMIT then
    aFrequencyLimit[siActArrayEntry].LimitDecrease := input;
  else
    CalcSimpleMode();
  end_if;
  if aFrequencyLimit[siActArrayEntry].LimitDecrease <> sWriteSDO.SDOData5.FrequLimitFalling2to4 then //do we have a new value?
    //Set new Limit
    sWriteSDO.SDOData5.FrequLimitFalling2to4 := aFrequencyLimit[siActArrayEntry].LimitDecrease;
    biReqSDOConfigRdWr.WriteConfigSDO5       := TRUE;
  end_if;

  result := FrequLimitDecrease2to4;

END_FUNCTION

FUNCTION VIRTUAL GLOBAL ST151Base::FrequLimitDecrease4to8::Write
	VAR_INPUT
		input (EAX) 	: UDINT;
	END_VAR
	VAR_OUTPUT
		result (EAX) 	: UDINT;
	END_VAR
  VAR
    siActArrayEntry : SINT;
  END_VAR

  siActArrayEntry := 2;
  //calculate compatibility mode if client is set
  input *= usCompModeVST;

   // Check for max frequency limit
  if input > ST151_MAXFREQUENCY_OUT then
    input := ST151_MAXFREQUENCY_OUT;
  end_if;
  //Save Input
  FrequLimitDecrease4to8 := input / usCompModeVST;

  if input <> ST151_AUTOSET_FREQUENCYLIMIT then
    aFrequencyLimit[siActArrayEntry].LimitDecrease := input;
  else
    CalcSimpleMode();
  end_if;
  if aFrequencyLimit[siActArrayEntry].LimitDecrease <> sWriteSDO.SDOData5.FrequLimitFalling4to8 then //do we have a new value?
    //Set new Limit
    sWriteSDO.SDOData5.FrequLimitFalling4to8 := aFrequencyLimit[siActArrayEntry].LimitDecrease;
    biReqSDOConfigRdWr.WriteConfigSDO5       := TRUE;
  end_if;

  result := FrequLimitDecrease4to8;

END_FUNCTION

FUNCTION VIRTUAL GLOBAL ST151Base::FrequLimitDecrease8to16::Write
	VAR_INPUT
		input (EAX) 	: UDINT;
	END_VAR
	VAR_OUTPUT
		result (EAX) 	: UDINT;
	END_VAR
  VAR
    siActArrayEntry : SINT;
  END_VAR

  siActArrayEntry := 3;
  //calculate compatibility mode if client is set
  input *= usCompModeVST;

   // Check for max frequency limit
  if input > ST151_MAXFREQUENCY_OUT then
    input := ST151_MAXFREQUENCY_OUT;
  end_if;
  //Save Input
  FrequLimitDecrease8to16 := input / usCompModeVST;

  if input <> ST151_AUTOSET_FREQUENCYLIMIT then
    aFrequencyLimit[siActArrayEntry].LimitDecrease := input;
  else
    CalcSimpleMode();
  end_if;
  if aFrequencyLimit[siActArrayEntry].LimitDecrease <> sWriteSDO.SDOData5.FrequLimitFalling8to16 then //do we have a new value?
    //Set new Limit
    sWriteSDO.SDOData5.FrequLimitFalling8to16 := aFrequencyLimit[siActArrayEntry].LimitDecrease;
    biReqSDOConfigRdWr.WriteConfigSDO5        := TRUE;
  end_if;

  result := FrequLimitDecrease8to16;

END_FUNCTION

FUNCTION VIRTUAL GLOBAL ST151Base::FrequLimitDecrease16to32::Write
	VAR_INPUT
		input (EAX) 	: UDINT;
	END_VAR
	VAR_OUTPUT
		result (EAX) 	: UDINT;
	END_VAR
  VAR
    siActArrayEntry : SINT;
  END_VAR

  siActArrayEntry := 4;
  //calculate compatibility mode if client is set
  input *= usCompModeVST;

   // Check for max frequency limit
  if input > ST151_MAXFREQUENCY_OUT then
    input := ST151_MAXFREQUENCY_OUT;
  end_if;
  //Save Input
  FrequLimitDecrease16to32 := input / usCompModeVST;

  if input <> ST151_AUTOSET_FREQUENCYLIMIT then
    aFrequencyLimit[siActArrayEntry].LimitDecrease := input;
  else
    CalcSimpleMode();
  end_if;
  if aFrequencyLimit[siActArrayEntry].LimitDecrease <> sWriteSDO.SDOData5.FrequLimitFalling16to32 then //do we have a new value?
    //Set new Limit
    sWriteSDO.SDOData5.FrequLimitFalling16to32 := aFrequencyLimit[siActArrayEntry].LimitDecrease;
    biReqSDOConfigRdWr.WriteConfigSDO5         := TRUE;
  end_if;

  result := FrequLimitDecrease16to32;

END_FUNCTION

FUNCTION VIRTUAL GLOBAL ST151Base::FrequLimitDecrease32to64::Write
	VAR_INPUT
		input (EAX) 	: UDINT;
	END_VAR
	VAR_OUTPUT
		result (EAX) 	: UDINT;
	END_VAR
  VAR
    siActArrayEntry : SINT;
  END_VAR

  siActArrayEntry := 5;
  //calculate compatibility mode if client is set
  input *= usCompModeVST;

   // Check for max frequency limit
  if input > ST151_MAXFREQUENCY_OUT then
    input := ST151_MAXFREQUENCY_OUT;
  end_if;
  //Save Input
  FrequLimitDecrease32to64 := input / usCompModeVST;

  if input <> ST151_AUTOSET_FREQUENCYLIMIT then
    aFrequencyLimit[siActArrayEntry].LimitDecrease := input;
  else
    CalcSimpleMode();
  end_if;
  if aFrequencyLimit[siActArrayEntry].LimitDecrease <> sWriteSDO.SDOData5.FrequLimitFalling32to64 then //do we have a new value?
    //Set new Limit
    sWriteSDO.SDOData5.FrequLimitFalling32to64 := aFrequencyLimit[siActArrayEntry].LimitDecrease;
    biReqSDOConfigRdWr.WriteConfigSDO5         := TRUE;
  end_if;

  result := FrequLimitDecrease32to64;

END_FUNCTION

FUNCTION ST151Base::CalcAdaptiveMicroStepping
	VAR_INPUT
		dTargetFrequency 	: DINT;
		dActSetFrequency 	: DINT;
	END_VAR
	VAR_OUTPUT
		dRetCode 	: DINT;
	END_VAR
  VAR
    usTempLimitCnt : USINT;
    bDesiredSteppingMode : BOOL;
    udActLowFrequency : UDINT;
    tempActiveSteps : bd_EnabledFreqLimit;
  END_VAR

  dRetCode          := 0;
  udActLowFrequency := 0;
  tempActiveSteps   := 0;
  bDesiredSteppingMode := FALSE;
  //search for needed steps
  if abs(dTargetFrequency) > abs(dActSetFrequency) then
    //acceleration
    sStepsNeeded.IncreaseFreq := 0;
    sAdaptiveStepping.usIncreaseActStepsActivated := 0;

    for usTempLimitCnt := 0  to ST151_MAXSTEPPING_MODES-1 do
      //step is needed if desired frequency is higher than frequency limit
      if abs(dTargetFrequency)$UDINT >= aFrequencyLimit[usTempLimitCnt].LimitIncrease then
        sStepsNeeded.IncreaseFreq := sStepsNeeded.IncreaseFreq or (1 shl (usTempLimitCnt));
        bDesiredSteppingMode      := TRUE;
        if abs(dActSetFrequency)$UDINT <= aFrequencyLimit[usTempLimitCnt].LimitIncrease then
          sStepsNeeded.IncreaseFreq := sStepsNeeded.IncreaseFreq or (1 shl (usTempLimitCnt+1));
        end_if;
      end_if;
    end_for;

    //activate 64 stepping mode if desired frequence is lower then this limit
    if bDesiredSteppingMode = FALSE then
      sStepsNeeded.IncreaseFreq := sStepsNeeded.IncreaseFreq or (1 shl usTempLimitCnt-1);
      sAdaptiveStepping.aIncreaseLimitsArrayEntry[sAdaptiveStepping.usIncreaseActStepsActivated] := usTempLimitCnt;
      sAdaptiveStepping.usIncreaseActStepsActivated += 1;
    else
      //delete bits if start frequence is higher than stepping mode
      for usTempLimitCnt := 0  to ST151_MAXSTEPPING_MODES do
        if abs(dActSetFrequency)$UDINT > aFrequencyLimit[usTempLimitCnt].LimitIncrease
        & (sStepsNeeded.IncreaseFreq shr usTempLimitCnt+1) and 0x01 then
          sStepsNeeded.IncreaseFreq := sStepsNeeded.IncreaseFreq xor (1 shl usTempLimitCnt+1);
        end_if;

        if (sStepsNeeded.IncreaseFreq shr usTempLimitCnt) and 0x01
        & (EnableSteps shr usTempLimitCnt) and 0x01 then
          sAdaptiveStepping.aIncreaseLimitsArrayEntry[sAdaptiveStepping.usIncreaseActStepsActivated] := usTempLimitCnt;
          sAdaptiveStepping.usIncreaseActStepsActivated += 1;
        end_if;
      end_for;
    end_if;

    //remove disabled steps
    sStepsNeeded.IncreaseFreq := sStepsNeeded.IncreaseFreq and EnableSteps;
    if sAdaptiveStepping.usIncreaseActStepsActivated > 2 then
      udActLowFrequency       := aFrequencyLimit[sAdaptiveStepping.aIncreaseLimitsArrayEntry[0]].LimitDecrease;
      //search for needed steppings for adaptive mode
      for usTempLimitCnt := 1 to sAdaptiveStepping.usIncreaseActStepsActivated-2 do
        if aFrequencyLimit[sAdaptiveStepping.aIncreaseLimitsArrayEntry[usTempLimitCnt]].LimitIncrease < udActLowFrequency then
          //step before must be activated
          tempActiveSteps := tempActiveSteps or (1 shl sAdaptiveStepping.aIncreaseLimitsArrayEntry[usTempLimitCnt]);
          udActLowFrequency := aFrequencyLimit[sAdaptiveStepping.aIncreaseLimitsArrayEntry[usTempLimitCnt]].LimitDecrease;
        end_if;
      end_for;
    end_if;
    //step for desired frequency is always needed
    tempActiveSteps := tempActiveSteps or (1 shl sAdaptiveStepping.aIncreaseLimitsArrayEntry[0]);
    //step of start frequency is always needed
    tempActiveSteps := tempActiveSteps or (1 shl sAdaptiveStepping.aIncreaseLimitsArrayEntry[sAdaptiveStepping.usIncreaseActStepsActivated-1]);

  else
    //decceleration
    sStepsNeeded.DecreaseFreq := 0;
    sAdaptiveStepping.usDecreaseActStepsActivated := 0;

    for usTempLimitCnt := 0  to ST151_MAXSTEPPING_MODES-1 do
      //step is needed if desired frequency is higher than frequency limit
      if abs(dActSetFrequency)$UDINT >= aFrequencyLimit[usTempLimitCnt].LimitIncrease then
        sStepsNeeded.DecreaseFreq := sStepsNeeded.DecreaseFreq or (1 shl usTempLimitCnt);
        bDesiredSteppingMode      := TRUE;
        if abs(dTargetFrequency)$UDINT <= aFrequencyLimit[usTempLimitCnt].LimitIncrease then
          sStepsNeeded.DecreaseFreq := sStepsNeeded.DecreaseFreq or (1 shl usTempLimitCnt+1);
        end_if;
      end_if;
    end_for;

    //activate 64 stepping mode if desired frequence is lower then this limit
    if bDesiredSteppingMode = FALSE then
      sStepsNeeded.DecreaseFreq := sStepsNeeded.DecreaseFreq or (1 shl usTempLimitCnt-1);
      sAdaptiveStepping.aDecreaseLimitsArrayEntry[sAdaptiveStepping.usDecreaseActStepsActivated] := usTempLimitCnt;
      sAdaptiveStepping.usDecreaseActStepsActivated += 1;
    else
      //delete bits if start frequence is higher than stepping mode
      for usTempLimitCnt := 0  to ST151_MAXSTEPPING_MODES do
        if abs(dTargetFrequency)$UDINT > aFrequencyLimit[usTempLimitCnt].LimitIncrease
        & (sStepsNeeded.DecreaseFreq shr usTempLimitCnt+1) and 0x01 then
          sStepsNeeded.DecreaseFreq := sStepsNeeded.DecreaseFreq xor (1 shl usTempLimitCnt+1);
        end_if;

        if (sStepsNeeded.DecreaseFreq shr usTempLimitCnt) and 0x01
        & (EnableSteps shr usTempLimitCnt) and 0x01 then
          sAdaptiveStepping.aDecreaseLimitsArrayEntry[sAdaptiveStepping.usDecreaseActStepsActivated] := usTempLimitCnt;
          sAdaptiveStepping.usDecreaseActStepsActivated += 1;
        end_if;
      end_for;
    end_if;

    //remove disabled steps
    sStepsNeeded.DecreaseFreq := sStepsNeeded.DecreaseFreq and EnableSteps;
    if sAdaptiveStepping.usDecreaseActStepsActivated > 2 then
      udActLowFrequency       := aFrequencyLimit[sAdaptiveStepping.aDecreaseLimitsArrayEntry[0]].LimitDecrease;
      //search for needed steppings for adaptive mode
      for usTempLimitCnt := 1 to sAdaptiveStepping.usDecreaseActStepsActivated-2 do
        if aFrequencyLimit[sAdaptiveStepping.aDecreaseLimitsArrayEntry[usTempLimitCnt]].LimitIncrease < udActLowFrequency then
          //step before must be activated
          tempActiveSteps := tempActiveSteps or (1 shl sAdaptiveStepping.aDecreaseLimitsArrayEntry[usTempLimitCnt]);
          udActLowFrequency := aFrequencyLimit[sAdaptiveStepping.aDecreaseLimitsArrayEntry[usTempLimitCnt]].LimitDecrease;
        end_if;
      end_for;
    end_if;
    //step for desired frequency is always needed
    tempActiveSteps := tempActiveSteps or (1 shl sAdaptiveStepping.aDecreaseLimitsArrayEntry[0]);
    //step of start frequency is always needed
    tempActiveSteps := tempActiveSteps or (1 shl sAdaptiveStepping.aDecreaseLimitsArrayEntry[sAdaptiveStepping.usDecreaseActStepsActivated-1]);

  end_if;

  //write activated steppings to module
  sAccesses.sWriteData.ControlWord.EnableFullStep  := tempActiveSteps.FullStep;
  sAccesses.sWriteData.ControlWord.EnableHalfStep  := tempActiveSteps.HalfStep;
  sAccesses.sWriteData.ControlWord.EnableStep4  := tempActiveSteps.MicroStepping4;
  sAccesses.sWriteData.ControlWord.EnableStep8  := tempActiveSteps.MicroStepping8;
  sAccesses.sWriteData.ControlWord.EnableStep16 := tempActiveSteps.MicroStepping16;
  sAccesses.sWriteData.ControlWord.EnableStep32 := tempActiveSteps.MicroStepping32;
  sAccesses.sWriteData.ControlWord.EnableStep64 := tempActiveSteps.MicroStepping64;

END_FUNCTION

FUNCTION VIRTUAL GLOBAL ST151Base::RefreshValues::Write
	VAR_INPUT
		input (EAX) 	: DINT;
	END_VAR
	VAR_OUTPUT
		result (EAX) 	: DINT;
	END_VAR

  if input <> RefreshValues then
    RefreshValues := input;
    case RefreshValues of
      0: //refreshing of values is deactivated

      1: //refresh values cyclic
//        biReqSDOConfigRdWr.ReadConfigSDO4 := TRUE;

      2: //refresh value one time
        biReqSDOConfigRdWr.ReadConfigSDO4 := TRUE;

    else
      //wrong value input
    end_case;

    result := RefreshValues;

  end_if;

END_FUNCTION

FUNCTION VIRTUAL GLOBAL ST151Base::EnableSteps::Write
	VAR_INPUT
		input (EAX) 	: ST151Base::bd_EnabledFreqLimit;
	END_VAR
	VAR_OUTPUT
		result (EAX) 	: ST151Base::bd_EnabledFreqLimit;
	END_VAR
  VAR
  	biControlWord  : t_ControlWord;
  END_VAR

  if EnableSteps <> input then
    if usCompModeVST = 2 then
      //deactivate microstep mode 64 if vst comp mode is active
      input.MicroStepping64 := 0;
    end_if;
    EnableSteps := input and 0x7F;
    //initialize variable
    biControlWord := sAccesses.sWriteData.ControlWord;
    biControlWord.EnableStep64 := EnableSteps.MicroStepping64; //
    biControlWord.EnableStep32 := EnableSteps.MicroStepping32; //
    biControlWord.EnableStep16 := EnableSteps.MicroStepping16; //
    biControlWord.EnableStep8  := EnableSteps.MicroStepping8; //
    biControlWord.EnableStep4  := EnableSteps.MicroStepping4; //
    biControlWord.EnableHalfStep := EnableSteps.HalfStep; //
    biControlWord.EnableFullStep := EnableSteps.FullStep := TRUE; // full step can not be deactivated!
    sAccesses.sWriteData.ControlWord := biControlWord;
    //calculate decrease steps again
    FrequLimitDecrease1to2.Write(input:=FrequLimitDecrease1to2);
    FrequLimitDecrease2to4.Write(input:=FrequLimitDecrease2to4);
    FrequLimitDecrease4to8.Write(input:=FrequLimitDecrease4to8);
    FrequLimitDecrease8to16.Write(input:=FrequLimitDecrease8to16);
    FrequLimitDecrease16to32.Write(input:=FrequLimitDecrease16to32);
    FrequLimitDecrease32to64.Write(input:=FrequLimitDecrease32to64);
  end_if;
	result := EnableSteps;

END_FUNCTION

FUNCTION VIRTUAL GLOBAL ST151Base::AddAccesses
	VAR_OUTPUT
		eModuleInitState 	: iprStates;
	END_VAR
  VAR
  	usTempCnt : USINT;
    uiTempLength : UINT;
  END_VAR

  eModuleInitState := READY;

  UseOszi := UseOszi.Read();

  if UseOszi then
    if AddWrAccess(hOffset              := ST151_OSZI_ADDR_WRITE
                 , uLength              := sizeof(t_s_OsziWrite)
                 , ppData               := #sAccessesOszi.pWriteHeader
                 , ppStateByte          := #sAccessesOszi.WriteHeaderControl.pStateByte
                 , ppControlByte        := #sAccessesOszi.WriteHeaderControl.pControlByte
                 , pAccessHandle        := #sAccessesOszi.WriteHeaderControl.AccessHandle
                 ) <> READY then
      LogError(pMsg:="@ZZZZ (ST151Base::AddAccesses) Adding write far memory access for oszi function failed! Update OS and/or fpga and/or SdiasManager-class.");
      //only deactivate oszi funktion
      UseOszi := 0;
      return;
    end_if;

    if AddRdAccess(hOffset              := ST151_OSZI_ADDR_READ
                 , uLength              := sizeof(t_s_OsziRead)
                 , ppData               := #sAccessesOszi.pReadHeader
                 , ppStateByte          := #sAccessesOszi.ReadHeaderControl.pStateByte
                 , ppControlByte        := #sAccessesOszi.ReadHeaderControl.pControlByte
                 , pAccessHandle        := #sAccessesOszi.ReadHeaderControl.AccessHandle
                 ) <> READY then
      LogError(pMsg:="@ZZZZ (ST151Base::AddAccesses) Adding read far memory access for oszi function failed! Update OS and/or fpga and/or SdiasManager-class.");
      //only deactivate oszi funktion
      UseOszi := 0;
      return;
    end_if;

    for usTempCnt := 0 to ST151_OSZI_MAX_PDOREAD-1 do
      uiTempLength := (usTempCnt+1)*ST151_OSZI_ONE_PDOSIZE;
      if uiTempLength > ST151_OSZI_BUFFER_SIZE then
        uiTempLength := ST151_OSZI_BUFFER_SIZE - (usTempCnt*ST151_OSZI_ONE_PDOSIZE);
      else
        uiTempLength := ST151_OSZI_ONE_PDOSIZE;
      end_if;

      if AddRdAccess(hOffset              := ST151_OSZI_ADDR_DATA + (sizeof(a_uiOsziValues)*usTempCnt)
                   , uLength              := uiTempLength
                   , ppData               := #sAccessesOszi.apOsziData[usTempCnt]
                   , ppStateByte          := #sAccessesOszi.aReadDataControl[usTempCnt].pStateByte
                   , ppControlByte        := #sAccessesOszi.aReadDataControl[usTempCnt].pControlByte
                   , pAccessHandle        := #sAccessesOszi.aReadDataControl[usTempCnt].AccessHandle
                   ) <> READY then
        LogError(pMsg:="@ZZZZ (ST151Base::AddAccesses) Adding read far memory access for oszi function failed! Update OS and/or fpga and/or SdiasManager-class.");
        //only deactivate oszi funktion
        UseOszi := 0;
        return;
      end_if;
    end_for;
  end_if;

END_FUNCTION

FUNCTION GLOBAL ST151Base::StartMeasure
	VAR_INPUT
		pData 	: ^void;
		uiTriggerLevel 	: UINT;
		uiSamplePrescaler 	: UINT;
		bStartStopMeasure 	: BOOL;
		usTriggerSetting 	: USINT;
		usTriggerOffset 	: USINT;
	END_VAR
	VAR_OUTPUT
		dRetCode 	: DINT;
	END_VAR

  dRetCode := 0;

  if UseOszi = 0 then
    dRetCode := -1;
    return;
  end_if;

  if pData = NIL then
    dRetCode := -2;
    return;
  end_if;

  sAccessesOszi.sWriteOszi.TriggerLevel        := uiTriggerLevel;
  sAccessesOszi.sWriteOszi.SampleTimePrescaler := uiSamplePrescaler;

  case usTriggerSetting of
    0:  sAccessesOszi.sWriteOszi.ControlOszi.RisingEdge  := TRUE;
        sAccessesOszi.sWriteOszi.ControlOszi.FallingEdge := FALSE;
        sAccessesOszi.sWriteOszi.ControlOszi.Force       := FALSE;

    1:  sAccessesOszi.sWriteOszi.ControlOszi.RisingEdge  := FALSE;
        sAccessesOszi.sWriteOszi.ControlOszi.FallingEdge := TRUE;
        sAccessesOszi.sWriteOszi.ControlOszi.Force       := FALSE;

    2:  sAccessesOszi.sWriteOszi.ControlOszi.RisingEdge  := FALSE;
        sAccessesOszi.sWriteOszi.ControlOszi.FallingEdge := FALSE;
        sAccessesOszi.sWriteOszi.ControlOszi.Force       := TRUE;
  else
    dRetCode := -3;
    return;
  end_case;

  case usTriggerOffset of
    0: sAccessesOszi.usOsziTriggerOffset := 0;
       sAccessesOszi.uiSamplesAfterTrigger := ST151_OSZI_MAX_SAMPLES;
       sAccessesOszi.uiSamplesBeforeTrigger  := 0;
    1: sAccessesOszi.usOsziTriggerOffset := 25;
       sAccessesOszi.uiSamplesAfterTrigger := ((ST151_OSZI_MAX_SAMPLES/4)*3);
       sAccessesOszi.uiSamplesBeforeTrigger  := (ST151_OSZI_MAX_SAMPLES/4);
    2: sAccessesOszi.usOsziTriggerOffset := 50;
       sAccessesOszi.uiSamplesAfterTrigger := (ST151_OSZI_MAX_SAMPLES/2);
       sAccessesOszi.uiSamplesBeforeTrigger  := (ST151_OSZI_MAX_SAMPLES/2);
    3: sAccessesOszi.usOsziTriggerOffset := 75;
       sAccessesOszi.uiSamplesAfterTrigger := (ST151_OSZI_MAX_SAMPLES/4);
       sAccessesOszi.uiSamplesBeforeTrigger  := ((ST151_OSZI_MAX_SAMPLES/4)*3);

  else
    dRetCode := -4;
    return;
  end_case;

  sAccessesOszi.sWriteOszi.SamplesAfterTrigger := sAccessesOszi.uiSamplesAfterTrigger-1;
  sAccessesOszi.bDataReady                     := FALSE;

  if bStartStopMeasure then
    if sAccessesOszi.eOsziData <> _OsziDataIdle then
      //other trigger is at progress
      dRetCode := -5;
      return;
    end_if;
    sAccessesOszi.pToExternData := pData;
    sAccessesOszi.sWriteOszi.ControlOszi.CancelTrigger   := FALSE;
    sAccessesOszi.sWriteOszi.ControlOszi.StartTriggering := TRUE;
    sAccessesOszi.bMeasureStarted                        := TRUE;
  else
    sAccessesOszi.sWriteOszi.ControlOszi.CancelTrigger   := TRUE;
    sAccessesOszi.sWriteOszi.ControlOszi.StartTriggering := FALSE;
    sAccessesOszi.bMeasureStarted                        := FALSE;
  end_if;
  //reset last oszi state
  sAccessesOszi.sLastOsziState.StateOszi := 0;
  sAccessesOszi.eOsziData := _OsziTriggerStart;

END_FUNCTION

FUNCTION ST151Base::GetMeasureData
	VAR_INPUT
		pData 	: ^void;
	END_VAR
  VAR
  	uiCopiedData : UINT;
  END_VAR

  uiCopiedData := 0;
  if sAccessesOszi.bSplitBuffer = FALSE then
    _memcpy(ptr1:=pData, ptr2:=sAccessesOszi.pFirstEntryOsziData, cntr:=sAccessesOszi.uiDatalength1);
  else
    //buffer data is splitted
    _memcpy(ptr1:=pData, ptr2:=sAccessesOszi.pFirstEntryOsziData, cntr:=sAccessesOszi.uiDatalength2);

    _memcpy(ptr1:=(pData+sAccessesOszi.uiDatalength2), ptr2:=#sAccessesOszi.aLastOsziData, cntr:=sAccessesOszi.uiDatalength1);
  end_if;

END_FUNCTION

FUNCTION GLOBAL ST151Base::GetMeasureState
	VAR_INPUT
		pbTriggered 	: ^BOOL;(* := NIL *)
	END_VAR
	VAR_OUTPUT
		dRetCode 	: DINT;
	END_VAR

  //get data is busy
  dRetCode := 1;

  if pbTriggered <> NIL then
    pbTriggered^ := sAccessesOszi.sLastOsziState.StateOszi.Triggered;
  end_if;

  if sAccessesOszi.bMeasureStarted = FALSE then
    dRetCode := -1;
    return;
  end_if;

  if sAccessesOszi.bDataReady then
    //data is available
    dRetCode := 0;
  end_if;

END_FUNCTION

FUNCTION GLOBAL ST151Base::GetActFreqLimits
	VAR_INPUT
		usValueIncDec 	: USINT;
		usArrayEntry 	: USINT;
		pusActCompMode 	: ^USINT;
	END_VAR
	VAR_OUTPUT
		udData 	: UDINT;
	END_VAR

  if usValueIncDec = 0 & usArrayEntry < ST151_MAXSTEPPING_MODES then
    udData := aFrequencyLimit[usArrayEntry].LimitIncrease;
  else
    udData := aFrequencyLimit[usArrayEntry].LimitDecrease;
  end_if;

  pusActCompMode^ := usCompModeVST;

END_FUNCTION

FUNCTION ST151Base::CalcSimpleMode
  VAR
    siTempCnt : SINT;
    udTempDecreaseLimit : UDINT;
    pFrequLimitData : ^UDINT;
    pSDOFrequLimit  : ^UDINT;
  END_VAR

  pFrequLimitData := #FrequLimitDecrease32to64.dData;
  pSDOFrequLimit  := #sWriteSDO.SDOData5.FrequLimitFalling32to64;
  udTempDecreaseLimit := 0;
  for siTempCnt := ST151_MAXSTEPPING_MODES-1 to 0 by -1 do
    if ((EnableSteps shr siTempCnt+1) and 0x01) = TRUE then
      udTempDecreaseLimit := aFrequencyLimit[siTempCnt].LimitIncrease;
      if udTempDecreaseLimit > udLimitsHysteresis  then
        udTempDecreaseLimit -= udLimitsHysteresis;
      else
        udTempDecreaseLimit := 0;
      end_if;
    end_if;
    //check if step is activated and limit is set to automatically
    if pFrequLimitData^ = 0
    & ((EnableSteps shr siTempCnt) and 0x01) = TRUE then
      aFrequencyLimit[siTempCnt].LimitDecrease := udTempDecreaseLimit;
    end_if;
    pSDOFrequLimit^ := aFrequencyLimit[siTempCnt].LimitDecrease;
    pFrequLimitData -= sizeof(SvrCh);
    pSDOFrequLimit += sizeof(UDINT);
  end_for;
  //write sdo data again for decreasing limits
  biReqSDOConfigRdWr.WriteConfigSDO5 := TRUE;

END_FUNCTION

FUNCTION VIRTUAL GLOBAL ST151Base::ChopperOffTime::Write
	VAR_INPUT
		input (EAX) 	: DINT;
	END_VAR
	VAR_OUTPUT
		result (EAX) 	: DINT;
	END_VAR

  if input < ST151_MIN_ALLOWED_CHOPPEROFFTIME then
    input := ST151_MIN_ALLOWED_CHOPPEROFFTIME;
  elsif input > ST151_MAX_ALLOWED_CHOPPEROFFTIME then
    input := ST151_MAX_ALLOWED_CHOPPEROFFTIME;
  end_if;

  ChopperOffTime := input;
  if ChopperOffTime <> sWriteSDO.SDOData1.ChopperOffTime then
    sWriteSDO.SDOData1.ChopperOffTime  := ChopperOffTime$UINT;
    biReqSDOConfigRdWr.WriteConfigSDO1 := TRUE;
  end_if;
	result := ChopperOffTime;

END_FUNCTION

FUNCTION VIRTUAL GLOBAL ST151Base::FastDecayTime::Write
	VAR_INPUT
		input (EAX) 	: DINT;
	END_VAR
	VAR_OUTPUT
		result (EAX) 	: DINT;
	END_VAR

  if input > ChopperOffTime then
    input := ChopperOffTime;
  elsif input < 0 then
    input := 0;
  end_if;

  FastDecayTime := input;
  if FastDecayTime <> sWriteSDO.SDOData1.FastDecayTime then
    sWriteSDO.SDOData1.FastDecayTime   := FastDecayTime$UINT;
    biReqSDOConfigRdWr.WriteConfigSDO1 := TRUE;
  end_if;
	result := FastDecayTime;

END_FUNCTION

FUNCTION VIRTUAL GLOBAL ST151Base::ChopperOnTimeMin::Write
	VAR_INPUT
		input (EAX) 	: DINT;
	END_VAR
	VAR_OUTPUT
		result (EAX) 	: DINT;
	END_VAR

  if input > ST151_MAX_ALLOWED_CHOPPEROFFTIME then
    input := ST151_MAX_ALLOWED_CHOPPEROFFTIME;
  elsif input < 0 then
    input := 0;
  end_if;

  ChopperOnTimeMin := input;
  if ChopperOffTime <> sWriteSDO.SDOData5.ChopperOnTimeMin then
    sWriteSDO.SDOData5.ChopperOnTimeMin  := ChopperOnTimeMin$UINT;
    biReqSDOConfigRdWr.WriteConfigSDO5 := TRUE;
  end_if;
	result := ChopperOnTimeMin;

END_FUNCTION

FUNCTION VIRTUAL GLOBAL ST151Base::FastDecayTimeFallingStep::Write
	VAR_INPUT
		input (EAX) 	: DINT;
	END_VAR
	VAR_OUTPUT
		result (EAX) 	: DINT;
	END_VAR

  if input > ChopperOffTime then
    input := ChopperOffTime;
  elsif input < 0 then
    input := 0;
  end_if;

  FastDecayTimeFallingStep := input;
  if FastDecayTimeFallingStep <> sWriteSDO.SDOData5.FastDecayTimeFallingStep then
    sWriteSDO.SDOData5.FastDecayTimeFallingStep := FastDecayTimeFallingStep$UINT;
    biReqSDOConfigRdWr.WriteConfigSDO5 := TRUE;
  end_if;
	result := FastDecayTimeFallingStep;

END_FUNCTION

FUNCTION VIRTUAL GLOBAL ST151Base::MaxCurrent::Write
	VAR_INPUT
		input (EAX) 	: DINT;
	END_VAR
	VAR_OUTPUT
		result (EAX) 	: DINT;
	END_VAR
  VAR
  	uiTmpReducedCurrent : UINT;
  END_VAR

  //Check Limit
  if input < 0 then
    input := 0;
  elsif input > ST151_MAX_ALLOWED_CURRENT then
    input := ST151_MAX_ALLOWED_CURRENT;
  end_if;

	MaxCurrent := input;
  uiTmpReducedCurrent := to_uint(MaxCurrent - ((MaxCurrent * StallCurrentReduction) / ST151_STALL_CURRENT_LIMIT));
  //check for changed values
  if MaxCurrent <> sWriteSDO.SDOData2.MaximumCurrentReg
  | uiTmpReducedCurrent <> sWriteSDO.SDOData2.ReducedCurrentReg then
    sWriteSDO.SDOData2.MaximumCurrentReg := MaxCurrent$UINT;
    sWriteSDO.SDOData2.ReducedCurrentReg := uiTmpReducedCurrent;
    biReqSDOConfigRdWr.WriteConfigSDO2 := TRUE;
  end_if;
	result := MaxCurrent;

END_FUNCTION

FUNCTION ST151Base::SetSDORdWrStep
	VAR_INPUT
		eActStep 	: t_e_SDOConfig;
	END_VAR
	VAR_OUTPUT
		eNextStep 	: t_e_SDOConfig;
	END_VAR
  VAR
  	biTmpActiveStep : t_bi_ReqSDOConfig;
  END_VAR

  case eActStep of
  	t_e_SDOConfig::_SDOConfig_Idle:   biTmpActiveStep := biReqSDOConfigRdWr;
  	t_e_SDOConfig::_SDOConfig_Write1: biTmpActiveStep := biReqSDOConfigRdWr and 0xFFFE;
  	t_e_SDOConfig::_SDOConfig_Write2: biTmpActiveStep := biReqSDOConfigRdWr and 0xFFFC;
  	t_e_SDOConfig::_SDOConfig_Write3: biTmpActiveStep := biReqSDOConfigRdWr and 0xFFF8;
  	t_e_SDOConfig::_SDOConfig_Write4: biTmpActiveStep := biReqSDOConfigRdWr and 0xFFF0;
  	t_e_SDOConfig::_SDOConfig_Write5: biTmpActiveStep := biReqSDOConfigRdWr and 0xFFE0;
  	t_e_SDOConfig::_SDOConfig_Write6: biTmpActiveStep := biReqSDOConfigRdWr and 0xFFC0;
  	t_e_SDOConfig::_SDOConfig_Read1: biTmpActiveStep := biReqSDOConfigRdWr and 0xFE00;
  	t_e_SDOConfig::_SDOConfig_Read2: biTmpActiveStep := biReqSDOConfigRdWr and 0xFC00;
  	t_e_SDOConfig::_SDOConfig_Read3: biTmpActiveStep := biReqSDOConfigRdWr and 0xF800;
  	t_e_SDOConfig::_SDOConfig_Read4: biTmpActiveStep := biReqSDOConfigRdWr and 0xF000;
  	t_e_SDOConfig::_SDOConfig_Read5: biTmpActiveStep := biReqSDOConfigRdWr and 0xC000;
  	t_e_SDOConfig::_SDOConfig_Read6: biTmpActiveStep := biReqSDOConfigRdWr and 0xE000;
  	t_e_SDOConfig::_SDOConfig_Finished:
  	t_e_SDOConfig::_SDOConfig_Error:
  end_case;

  if biTmpActiveStep.WriteConfigSDO1 then
    eNextStep  := _SDOConfig_Write1;
  elsif biTmpActiveStep.WriteConfigSDO2 then
    eNextStep  := _SDOConfig_Write2;
  elsif biTmpActiveStep.WriteConfigSDO3 then
    eNextStep  := _SDOConfig_Write3;
  elsif biTmpActiveStep.WriteConfigSDO4 then
    eNextStep  := _SDOConfig_Write4;
  elsif biTmpActiveStep.WriteConfigSDO5 then
    eNextStep  := _SDOConfig_Write5;
  elsif biTmpActiveStep.WriteConfigSDO6 then
    eNextStep  := _SDOConfig_Write6;
  elsif biTmpActiveStep.ReadConfigSDO1 then
    eNextStep  := _SDOConfig_Read1;
  elsif biTmpActiveStep.ReadConfigSDO2 then
    eNextStep  := _SDOConfig_Read2;
  elsif biTmpActiveStep.ReadConfigSDO3 then
    eNextStep  := _SDOConfig_Read3;
  elsif biTmpActiveStep.ReadConfigSDO4 then
    eNextStep  := _SDOConfig_Read4;
  elsif biTmpActiveStep.ReadConfigSDO5 then
    eNextStep  := _SDOConfig_Read5;
  elsif biTmpActiveStep.ReadConfigSDO6 then
    eNextStep  := _SDOConfig_Read6;
  else
    eNextStep  := _SDOConfig_Finished;
  end_if;

END_FUNCTION

FUNCTION VIRTUAL GLOBAL ST151Base::CurrentOffsetAdjBridge1::Write
	VAR_INPUT
		input (EAX) 	: DINT;
	END_VAR
	VAR_OUTPUT
		result (EAX) 	: DINT;
	END_VAR

  if input > ST151_CURRENTOFFSETADJUST_MAX then
    input := ST151_CURRENTOFFSETADJUST_MAX;
  elsif input < ST151_CURRENTOFFSETADJUST_MIN then
    input := ST151_CURRENTOFFSETADJUST_MIN;
  end_if;

  CurrentOffsetAdjBridge1 := input;
  if CurrentOffsetAdjBridge1 <> sWriteSDO.SDOData6.CurrentOffsetAdjBridge1 then
    sWriteSDO.SDOData6.CurrentOffsetAdjBridge1 := CurrentOffsetAdjBridge1$INT;
    biReqSDOConfigRdWr.WriteConfigSDO6 := TRUE;
  end_if;
	result := CurrentOffsetAdjBridge1;

END_FUNCTION

FUNCTION VIRTUAL GLOBAL ST151Base::CurrentOffsetAdjBridge2::Write
	VAR_INPUT
		input (EAX) 	: DINT;
	END_VAR
	VAR_OUTPUT
		result (EAX) 	: DINT;
	END_VAR

  if input > ST151_CURRENTOFFSETADJUST_MAX then
    input := ST151_CURRENTOFFSETADJUST_MAX;
  elsif input < ST151_CURRENTOFFSETADJUST_MIN then
    input := ST151_CURRENTOFFSETADJUST_MIN;
  end_if;

  CurrentOffsetAdjBridge2 := input;
  if CurrentOffsetAdjBridge2 <> sWriteSDO.SDOData6.CurrentOffsetAdjBridge2 then
    sWriteSDO.SDOData6.CurrentOffsetAdjBridge2 := CurrentOffsetAdjBridge2$INT;
    biReqSDOConfigRdWr.WriteConfigSDO6 := TRUE;
  end_if;
	result := CurrentOffsetAdjBridge2;

END_FUNCTION
